// TIA Portal V17 export
// export: Created 2022-03-12T16:05:32.8701099Z, ExportSetting WithDefaults, DisplayName Totally Integrated Automation Portal, DisplayVersion V17, DisplayName TIA Portal Openness, DisplayVersion V17, DisplayName TIA Portal Version Control Interface, DisplayVersion V17, DisplayName STEP 7 Professional, DisplayVersion V17, DisplayName STEP 7 Safety, DisplayVersion V17, DisplayName WinCC Advanced / Unified PC, DisplayVersion V17
TYPE "CPG_typeEventCfg"
// stored: IsFailsafeCompliant false
   STRUCT
      ID : Int;   // ID Value - from PackTags Reason Code, 1=E-Stop pushed, 3=Main off, etc.
      value : Int;   // Reason Code 'Value' - allows for detailed breakdown of ID, ie 1=Discharge,
      message : Array[0.."LPMLV30_LANGUAGES_UPPER_LIM"] of String[60];   // Alarm Message - 0=English, 1=German, 2=Spanish, 3=Italian, 4=French
      category : Int;   // Category Value (0-9)
   END_STRUCT;
END_TYPE
